SUBAPPLICATION Ventilsteuerung_Uebung_023 (* Spiegelabfolge (3) *)
  (* Standard: 61499-2 *)
  (* Version 1.0, 2023-10-23, franz *)
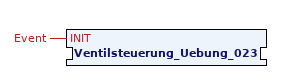
  EVENT_INPUT
    INIT;
  END_EVENT
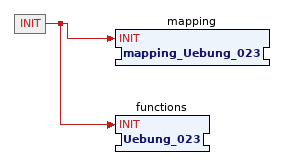
  SUBAPPS
    mapping : mapping_Uebung_023;
    functions : Uebung_023;
  END_SUBAPPS
  EVENT_CONNECTIONS
    INIT TO functions.INIT;
    INIT TO mapping.INIT;
  END_CONNECTIONS
END_SUBAPPLICATION
